{attribute 'GeneratedUsingTerminal: EL2819-0000-0016'}
{attribute addProperty BoxType "EL2819-0000-0016"}
{attribute addProperty Id "EtcSlaveTerminalBaseDIG_Diag_InputsAT %I*DIG_Diag_Inputs_F289D61564DIG_Inputs_DeviceAT %I*DIG_Inputs_Device_A1F150A94DIG_OutputsAT %Q*DIG_Outputs_B9300CB616WcStateAT %I*WcState_9091E0EB2InfoDataAT %I*InfoData_32EB74EA10"}
{attribute addProperty CRC "2879627376"}
{attribute addProperty Size "96"}
TYPE EL2819_ABA3A070 EXTENDS EtcSlaveTerminalBase :
STRUCT
	{attribute addProperty Name "DIG_Diag_Inputs"}
	DIG_Diag_Inputs : DIG_Diag_Inputs_F289D615;
	{attribute addProperty Name "DIG_Inputs_Device"}
	DIG_Inputs_Device : DIG_Inputs_Device_A1F150A9;
	{attribute addProperty Name "DIG_Outputs"}
	DIG_Outputs : DIG_Outputs_B9300CB6;
	{attribute addProperty Name "WcState"}
	WcState : WcState_9091E0EB;
	{attribute addProperty Name "InfoData"}
	InfoData : InfoData_32EB74EA;
END_STRUCT
END_TYPE

(* stored: Version 1.2.0.0, ProductVersion 3.1.4024.9
   DUT EL2819_ABA3A070: Id {cd9e6c09-8809-4712-b537-5f4547227c5f} *)
